{attribute 'GeneratedUsingTerminal: EL6201-0000-0017'}
{attribute addProperty BoxType "EL6201-0000-0017"}
{attribute addProperty Id "Slave_12A_DI0BOOL1Slave_12A_DI1BOOL1Slave_12A_DI2BOOL1Slave_12A_DI3BOOL1Slave_12B_DI0BOOL1Slave_12B_DI1BOOL1Slave_12B_DI2BOOL1Slave_12B_DI3BOOL1"}
{attribute addProperty CRC "2718058526"}
{attribute addProperty Size "8"}
TYPE Slave_12_Inputs_A202481E :
STRUCT
	{attribute addProperty Name "Slave_12A_DI0"}
	Slave_12A_DI0 : BOOL;
	{attribute addProperty Name "Slave_12A_DI1"}
	Slave_12A_DI1 : BOOL;
	{attribute addProperty Name "Slave_12A_DI2"}
	Slave_12A_DI2 : BOOL;
	{attribute addProperty Name "Slave_12A_DI3"}
	Slave_12A_DI3 : BOOL;
	{attribute addProperty Name "Slave_12B_DI0"}
	Slave_12B_DI0 : BOOL;
	{attribute addProperty Name "Slave_12B_DI1"}
	Slave_12B_DI1 : BOOL;
	{attribute addProperty Name "Slave_12B_DI2"}
	Slave_12B_DI2 : BOOL;
	{attribute addProperty Name "Slave_12B_DI3"}
	Slave_12B_DI3 : BOOL;
END_STRUCT
END_TYPE

(* stored: Version 1.2.0.0, ProductVersion 3.1.4024.11
   DUT Slave_12_Inputs_A202481E: Id {db0a967c-33ee-4df5-a8c3-42b82d60e45c} *)
